// TIA Portal V18 export
DATA_BLOCK "gDb_IO"   // DB20
{ S7_Optimized_Access := 'TRUE' }
VERSION : 0.1
// stored: AutoNumber true, DBAccessibleFromOPCUA true, DBAccessibleFromWebserver true, IsOnlyStoredInLoadMemory false, IsRetainMemResEnabled false, IsWriteProtectedInAS false, MemoryReserve 100
   VAR
      Andon1 : "UDT_andonIO";
      Andon2 : "UDT_andonIO";
      Andon3 : "UDT_andonIO";
      Andon4 : "UDT_andonIO";
      Andon5 : "UDT_andonIO";
      Andon6 : "UDT_andonIO";
      Andon7 : "UDT_andonIO";
      Andon8 : "UDT_andonIO";
      Andon9 : "UDT_andonIO";
      Andon10 : "UDT_andonIO";
      Sirene { S7_SetPoint := 'True'} : "UDT_sireneIO";
      SignalColumn { S7_SetPoint := 'True'} : "UDT_signalColumn";
      NokButton1 { S7_SetPoint := 'True'} : "UDT_nokButtonIO";
      NokButton2 { S7_SetPoint := 'True'} : "UDT_nokButtonIO";
      I_PartProduced { S7_SetPoint := 'True'} : Bool;
   END_VAR
BEGIN
END_DATA_BLOCK
